{attribute 'GeneratedUsingTerminal: EP5101-0011-0016'}
{attribute addProperty BoxType "EP5101-0011-0016"}
{attribute addProperty Id "ControlAT %Q*Control_6EF2C5D04Set_counter_valueAT %Q*UINT2"}
{attribute addProperty CRC "568512845"}
{attribute addProperty Size "6"}
TYPE ENC_Control_compact_21E2D14D :
STRUCT
	{attribute addProperty Name "Control"}
	Control AT %Q* : Control_6EF2C5D0;
	{attribute addProperty Name "Set_counter_value"}
	Set_counter_value AT %Q* : UINT;
END_STRUCT
END_TYPE

(* stored: Version 1.2.0.0, ProductVersion 3.1.4024.9
   DUT ENC_Control_compact_21E2D14D: Id {8ad49a4d-8505-4927-b236-b486768d03ee} *)
